// TIA Portal V16 export
// export: Created 2021-07-03T21:22:42.2990568Z, ExportSetting WithDefaults, DisplayName Totally Integrated Automation Portal, DisplayVersion V16, DisplayName TIA Portal Version Control Interface, DisplayVersion V16, DisplayName TIA Portal Openness, DisplayVersion V16, DisplayName STEP 7 Professional, DisplayVersion V16, DisplayName STEP 7 Safety, DisplayVersion V16, DisplayName WinCC Professional, DisplayVersion V16
TYPE "ConfigIF_MPLC_to_Plant"
// stored: IsFailsafeCompliant false
   STRUCT
      Spare_1 { ExternalAccessible := 'False'; ExternalVisible := 'False'; ExternalWritable := 'False'} : Word;   // Machine Features (refer to the Standard Machine Configuration Data)
      Machine_Product_ID { ExternalAccessible := 'False'; ExternalVisible := 'False'; ExternalWritable := 'False'} : Byte;   // Machine Product ID (refer to the Standard Machine Configuration Data)
      Machine_SortFraction { ExternalAccessible := 'False'; ExternalVisible := 'False'; ExternalWritable := 'False'} : Byte;   // Machine Sort Fraction (refer to the Standard Machine Configuration Data)
      Machine_Function { ExternalAccessible := 'False'; ExternalVisible := 'False'; ExternalWritable := 'False'} : Byte;   // Machine Function (refer to the Standard Machine Configuration Data)
      Machine_Cluster_ID { ExternalAccessible := 'False'; ExternalVisible := 'False'; ExternalWritable := 'False'} : Byte;   // Machine Cluster number (0-255)
      Machine_Cluster_Configuration { ExternalAccessible := 'False'; ExternalVisible := 'False'; ExternalWritable := 'False'} : Word;   // Machine Cluster Configuration (refer to the Standard Machine Configuration Data)
      PCS_PrimaryProtocol { ExternalAccessible := 'False'; ExternalVisible := 'False'; ExternalWritable := 'False'} : Byte;   // Primary Plant communication Protocol (Refer to Standard Machine Configuration Document)
      PCS_SecondaryProtocol { ExternalAccessible := 'False'; ExternalVisible := 'False'; ExternalWritable := 'False'} : Byte;   // Secondary Plant communication Protocol (Refer to Standard Machine Configuration Document)
      Hardware_Configuration_ID { ExternalAccessible := 'False'; ExternalVisible := 'False'; ExternalWritable := 'False'} : Byte;   // Machine PLC hardware configuration option (0-255)
      OPC_UA_ControlClient { ExternalAccessible := 'False'; ExternalVisible := 'False'; ExternalWritable := 'False'} : Bool;   // 0= Control Client Disabled; 1=Control Client Enabled
      OPC_UA_ViewClient_1 { ExternalAccessible := 'False'; ExternalVisible := 'False'; ExternalWritable := 'False'} : Bool;   // 0= View Client 1 Disabled; 1=View Client 1 Enabled
      OPC_UA_ViewClient_2 { ExternalAccessible := 'False'; ExternalVisible := 'False'; ExternalWritable := 'False'} : Bool;   // 0= View Client 2 Disabled; 1=View Client 2 Enabled
      OPC_UA_ViewClient_3 { ExternalAccessible := 'False'; ExternalVisible := 'False'; ExternalWritable := 'False'} : Bool;   // 0= View Client 3 Disabled; 1=View Client 3 Enabled
      Spare11_4 { ExternalAccessible := 'False'; ExternalVisible := 'False'; ExternalWritable := 'False'} : Bool;   // Reserved spare
      Spare11_5 { ExternalAccessible := 'False'; ExternalVisible := 'False'; ExternalWritable := 'False'} : Bool;   // Reserved spare
      Spare11_6 { ExternalAccessible := 'False'; ExternalVisible := 'False'; ExternalWritable := 'False'} : Bool;   // Reserved spare
      Spare11_7 { ExternalAccessible := 'False'; ExternalVisible := 'False'; ExternalWritable := 'False'} : Bool;   // Reserved spare
      Machine_IP_Address { ExternalAccessible := 'False'; ExternalVisible := 'False'; ExternalWritable := 'False'} : Array[1..4] of Byte;   // Machine PLC IP address (xx-xx-xx-xx)
      Machine_TCP_Port { ExternalAccessible := 'False'; ExternalVisible := 'False'; ExternalWritable := 'False'} : Int;   // Machine PLC TCP port number (2010-5000)
      Machine_TSAP { ExternalAccessible := 'False'; ExternalVisible := 'False'; ExternalWritable := 'False'} : Array[1..16] of Byte;   // Machine PLC TSAP (string containing Machine to 16 x ASCII characters)
      Machine_MAC_Address { ExternalAccessible := 'False'; ExternalVisible := 'False'; ExternalWritable := 'False'} : Array[0..5] of Byte;   // Machine PLC MAC address (xx-xx-xx-xx-xx-xx)
      Plant_Connection_ID { ExternalAccessible := 'False'; ExternalVisible := 'False'; ExternalWritable := 'False'} : Int;   // Plant PLC connection reference (1-65535)
      Spare { ExternalAccessible := 'False'; ExternalVisible := 'False'; ExternalWritable := 'False'} : Int;   // Reserved spare
      NTP_Server_IP_Address { ExternalAccessible := 'False'; ExternalVisible := 'False'; ExternalWritable := 'False'} : Array[1..4] of Byte;   // NTP Time Server Address (xx-xx-xx-xx)
      Last_PCS_Config_Hours { ExternalAccessible := 'False'; ExternalVisible := 'False'; ExternalWritable := 'False'} : Byte;   // Last configuration date/time recorded on the PLC after PCS config request from OTI or Plant. OTI/SCADA username transferred by PLC (depending on the config source)
      Last_PCS_Config_Minutes { ExternalAccessible := 'False'; ExternalVisible := 'False'; ExternalWritable := 'False'} : Byte;   // As above
      Last_PCS_Config_Century { ExternalAccessible := 'False'; ExternalVisible := 'False'; ExternalWritable := 'False'} : Byte;   // As above
      Last_PCS_Config_Year { ExternalAccessible := 'False'; ExternalVisible := 'False'; ExternalWritable := 'False'} : Byte;   // As above
      Last_PCS_Config_Month { ExternalAccessible := 'False'; ExternalVisible := 'False'; ExternalWritable := 'False'} : Byte;   // As above
      Last_PCS_Config_Day { ExternalAccessible := 'False'; ExternalVisible := 'False'; ExternalWritable := 'False'} : Byte;   // As above
      UserName { ExternalAccessible := 'False'; ExternalVisible := 'False'; ExternalWritable := 'False'} : Array[0..7] of Byte;   // Name of user (SCADA or OTI), who performed PCS configuration
      PCS_Config_Source { ExternalAccessible := 'False'; ExternalVisible := 'False'; ExternalWritable := 'False'} : Byte;   // PCS Configuration source: 0 - None; 1 - OTI; 2 - Plant
      OPC_UA_ControlClient_Active { ExternalAccessible := 'False'; ExternalVisible := 'False'; ExternalWritable := 'False'} : Bool;   // 1=OPC-UA ControlClient Active; 0=OPC-UA ControlClient Inactive
      OPC_UA_ViewClient_1_Active { ExternalAccessible := 'False'; ExternalVisible := 'False'; ExternalWritable := 'False'} : Bool;   // 1=OPC-UA ViewClient_1 Active; 0=OPC-UA ViewClient_1 Inactive
      OPC_UA_ViewClient_2_Active { ExternalAccessible := 'False'; ExternalVisible := 'False'; ExternalWritable := 'False'} : Bool;   // 1=OPC-UA ViewClient_2 Active; 0=OPC-UA ViewClient_2 Inactive
      OPC_UA_ViewClient_3_Active { ExternalAccessible := 'False'; ExternalVisible := 'False'; ExternalWritable := 'False'} : Bool;   // 1=OPC-UA ViewClient_3 Active; 0=OPC-UA ViewClient_3 Inactive
      Spare63_4 { ExternalAccessible := 'False'; ExternalVisible := 'False'; ExternalWritable := 'False'} : Bool;   // Reserved spare
      Spare63_5 { ExternalAccessible := 'False'; ExternalVisible := 'False'; ExternalWritable := 'False'} : Bool;   // Reserved spare
      Primary_Protocol_Comms_OK { ExternalAccessible := 'False'; ExternalVisible := 'False'; ExternalWritable := 'False'} : Bool;   // Plant Control Network Communication Status (0=Error; 1=OK)
      Secondary_Protocol_Comms_OK { ExternalAccessible := 'False'; ExternalVisible := 'False'; ExternalWritable := 'False'} : Bool;   // Plant SMachineervision Network Communication Status (0=Error; 1=OK)
      OPC_UA_PortNumber { ExternalAccessible := 'False'; ExternalVisible := 'False'; ExternalWritable := 'False'} : UInt;   // Machine- configured OPC-UA port
      Profibus_Address { ExternalAccessible := 'False'; ExternalVisible := 'False'; ExternalWritable := 'False'} : Byte;   // Machine- configured Profibus Address
      Spare67 { ExternalAccessible := 'False'; ExternalVisible := 'False'; ExternalWritable := 'False'} : Byte;   // Reserved spare
      Spare68 { ExternalAccessible := 'False'; ExternalVisible := 'False'; ExternalWritable := 'False'} : Byte;   // Reserved spare
      Spare69 { ExternalAccessible := 'False'; ExternalVisible := 'False'; ExternalWritable := 'False'} : Byte;   // Reserved spare
      Spare70 { ExternalAccessible := 'False'; ExternalVisible := 'False'; ExternalWritable := 'False'} : Byte;   // Reserved spare
      Spare71 { ExternalAccessible := 'False'; ExternalVisible := 'False'; ExternalWritable := 'False'} : Byte;   // Reserved spare
      Spare72 { ExternalAccessible := 'False'; ExternalVisible := 'False'; ExternalWritable := 'False'} : Byte;   // Reserved spare
      Spare73 { ExternalAccessible := 'False'; ExternalVisible := 'False'; ExternalWritable := 'False'} : Byte;   // Reserved spare
      Spare74 { ExternalAccessible := 'False'; ExternalVisible := 'False'; ExternalWritable := 'False'} : Byte;   // Reserved spare
      Spare75 { ExternalAccessible := 'False'; ExternalVisible := 'False'; ExternalWritable := 'False'} : Byte;   // Reserved spare
      Spare76 { ExternalAccessible := 'False'; ExternalVisible := 'False'; ExternalWritable := 'False'} : Byte;   // Reserved spare
      Spare77 { ExternalAccessible := 'False'; ExternalVisible := 'False'; ExternalWritable := 'False'} : Byte;   // Reserved spare
      Spare78 { ExternalAccessible := 'False'; ExternalVisible := 'False'; ExternalWritable := 'False'} : Byte;   // Reserved spare
      Spare79 { ExternalAccessible := 'False'; ExternalVisible := 'False'; ExternalWritable := 'False'} : Byte;   // Reserved spare
      Spare80 { ExternalAccessible := 'False'; ExternalVisible := 'False'; ExternalWritable := 'False'} : Byte;   // Reserved spare
      Spare81 { ExternalAccessible := 'False'; ExternalVisible := 'False'; ExternalWritable := 'False'} : Byte;   // Reserved spare
      Spare82 { ExternalAccessible := 'False'; ExternalVisible := 'False'; ExternalWritable := 'False'} : Byte;   // Reserved spare
      Spare83 { ExternalAccessible := 'False'; ExternalVisible := 'False'; ExternalWritable := 'False'} : Byte;   // Reserved spare
      Spare84 { ExternalAccessible := 'False'; ExternalVisible := 'False'; ExternalWritable := 'False'} : Byte;   // Reserved spare
      Spare85 { ExternalAccessible := 'False'; ExternalVisible := 'False'; ExternalWritable := 'False'} : Byte;   // Reserved spare
      Spare86 { ExternalAccessible := 'False'; ExternalVisible := 'False'; ExternalWritable := 'False'} : Byte;   // Reserved spare
      Spare87 { ExternalAccessible := 'False'; ExternalVisible := 'False'; ExternalWritable := 'False'} : Byte;   // Reserved spare
      Spare88 { ExternalAccessible := 'False'; ExternalVisible := 'False'; ExternalWritable := 'False'} : Byte;   // Reserved spare
      Spare89 { ExternalAccessible := 'False'; ExternalVisible := 'False'; ExternalWritable := 'False'} : Byte;   // Reserved spare
      Machine_Features { ExternalAccessible := 'False'; ExternalVisible := 'False'; ExternalWritable := 'False'} : DWord;   // Machine Features (refer to the Standard Machine Configuration Data)
      Machine_Features_Mask { ExternalAccessible := 'False'; ExternalVisible := 'False'; ExternalWritable := 'False'} : DWord;   // Machine Features Mask (refer to the Standard Machine Configuration Data)
      OTI_CheckCycle_Override_Control_State { ExternalAccessible := 'False'; ExternalVisible := 'False'; ExternalWritable := 'False'} : Bool;   // 1 = 'Override Checkercycle' control on OTI Disabled
      OTI_Configuration_Control_Status { ExternalAccessible := 'False'; ExternalVisible := 'False'; ExternalWritable := 'False'} : Bool;   // 1 = OTI PCS Configuration Machinedate button disabled
      OTI_PCS_Config { ExternalAccessible := 'False'; ExternalVisible := 'False'; ExternalWritable := 'False'} : Bool;   // Configuration pulse from OTI (pulsed for 1sec)
      OTI_Authentication_Mode { ExternalAccessible := 'False'; ExternalVisible := 'False'; ExternalWritable := 'False'} : Bool;   // Machine user authentication mode (0=password; 1= biometrics)
      Machine_Init { ExternalAccessible := 'False'; ExternalVisible := 'False'; ExternalWritable := 'False'} : Bool;   // PLC IP Address /HW Config Machinedate pulse (pulsed for 1sec)
      OTI_Ej_Sense_Feedback_Control_State { ExternalAccessible := 'False'; ExternalVisible := 'False'; ExternalWritable := 'False'} : Bool;   // 1 = 'Override Ejector Sense Feedback Alarms' on OTI disabled
      Spare98_6 { ExternalAccessible := 'False'; ExternalVisible := 'False'; ExternalWritable := 'False'} : Bool;   // Reserved spare
      TimeSync_Source { ExternalAccessible := 'False'; ExternalVisible := 'False'; ExternalWritable := 'False'} : Bool;   // Time Synchronization Source (0=NTP Server; 1= Interface DB)
      Spare99_0 { ExternalAccessible := 'False'; ExternalVisible := 'False'; ExternalWritable := 'False'} : Bool;   // Reserved spare
      Spare99_1 { ExternalAccessible := 'False'; ExternalVisible := 'False'; ExternalWritable := 'False'} : Bool;   // Reserved spare
      Spare99_2 { ExternalAccessible := 'False'; ExternalVisible := 'False'; ExternalWritable := 'False'} : Bool;   // Reserved spare
      Spare99_3 { ExternalAccessible := 'False'; ExternalVisible := 'False'; ExternalWritable := 'False'} : Bool;   // Reserved spare
      Spare99_4 { ExternalAccessible := 'False'; ExternalVisible := 'False'; ExternalWritable := 'False'} : Bool;   // Reserved spare
      Spare99_5 { ExternalAccessible := 'False'; ExternalVisible := 'False'; ExternalWritable := 'False'} : Bool;   // Reserved spare
      Spare99_6 { ExternalAccessible := 'False'; ExternalVisible := 'False'; ExternalWritable := 'False'} : Bool;   // Reserved spare
      PCS_Config_Machinedate_Done { ExternalAccessible := 'False'; ExternalVisible := 'False'; ExternalWritable := 'False'} : Bool;   // 1 sec Confirmation pulse – configuration date, time and username recorded in the event log
   END_STRUCT;
END_TYPE
